// TIA Portal project "Deliverable_1" (V17)

(* hardware
DEVICE "S7-1200 station_1"  S7-1200 Station
   slot 0: "Rack_0"  S7-1200 Rack  Rack  V1.0
   slot 1: "PLC_1"  CPU 1217C DC/DC/DC  6ES7 217-1AG40-0XB0  V4.5
*)

// ===== PLC "PLC_1"  CPU 1217C DC/DC/DC =====

VAR_GLOBAL   // PLC tag table "Default tag table"
   "Start_Push_Button" AT %I0.0 : Bool;
   "Reset_Button" AT %I0.1 : Bool;
   "Elapsed_Time" AT %MD0 : Time;
   "Motor" AT %Q0.0 : Bool;
   "Motor_Memory" AT %M0.1 : Bool;
END_VAR

// folder: System blocks/Program resources

DATA_BLOCK "IEC_Timer_0_DB"   // DB1
{ S7_Optimized_Access := 'TRUE' }
AUTHOR : Simatic
FAMILY : IEC
NAME : IEC_TMR
VERSION : 1.0
// stored: InstanceOfName IEC_TIMER
"IEC_TIMER"
BEGIN
END_DATA_BLOCK

// folder: (top level)

ORGANIZATION_BLOCK "Main"   // OB1, LAD, ProgramCycle
TITLE = "Main Program Sweep (Cycle)"
{ S7_Optimized_Access := 'TRUE' }
VERSION : 0.1
   VAR_INPUT
      Initial_Call : Bool;   // Initial call of this OB
      Remanence : Bool;   // =True, if remanent data are available
   END_VAR
BEGIN

REGION Network 1
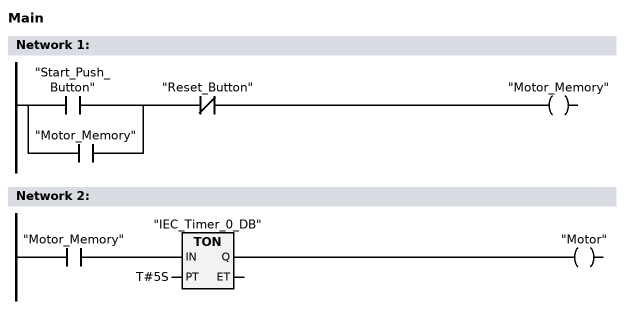
   RUNG wire#powerrail
      Contact( "Start_Push_Button" )
      wire#w1
      I_Contact( "Reset_Button" )
      Coil( "Motor_Memory" )
   END_RUNG
   RUNG wire#powerrail
      Contact( "Motor_Memory" )
   END_RUNG wire#w1
   // the same network as SCL:
   "Motor_Memory" := ("Start_Push_Button" OR "Motor_Memory") AND NOT "Reset_Button";
END_REGION

REGION Network 2
   "IEC_Timer_0_DB".TON(IN := "Motor_Memory", PT := T#5S);
   "Motor" := "IEC_Timer_0_DB".Q;
END_REGION
END_ORGANIZATION_BLOCK